FUNCTION_BLOCK GROUPING
  {SET_ATTRIBUTE(OpcUa, SERVICE)}
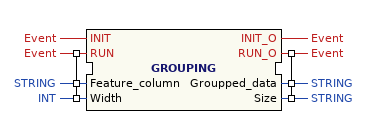
  EVENT_INPUT
    INIT;
    RUN WITH Feature_column, Width; {SET_ATTRIBUTE(OpcUa, Method)}
  END_EVENT
  EVENT_OUTPUT
    INIT_O;
    RUN_O WITH Groupped_data, Size;
  END_EVENT
  VAR_INPUT
    Feature_column : STRING; {SET_ATTRIBUTE(OpcUa, Variable.RUN)}
    Width : INT; {SET_ATTRIBUTE(OpcUa, Variable.RUN)}
  END_VAR
  VAR_OUTPUT
    Groupped_data : STRING; {SET_ATTRIBUTE(OpcUa, Variable.RUN)}
    Size : STRING; {SET_ATTRIBUTE(OpcUa, Variable.RUN)}
  END_VAR
END_FUNCTION_BLOCK
